# EPICS substitutions: ethmodApp/Db/AKI2C_AD527x.substitutions
file AKI2C_AD527x_dev.template
{
   pattern { P    ,R    ,PORT    ,ADDR     ,TIMEOUT     }
           { $(P) ,$(R) ,$(PORT) ,$(ADDR)  ,$(TIMEOUT)  }
}
